// TwinCAT 3 PLC project PLC_to_Cpp
// ProgramVersion: 3.1.4023.0
// libraries:
//   Tc2_Standard, * (Beckhoff Automation GmbH)
//   Tc2_System, * (Beckhoff Automation GmbH)
//   Tc2_Utilities, * (Beckhoff Automation GmbH)
//   Tc3_IotBase, * (Beckhoff Automation GmbH)
//   Tc3_Module, * (Beckhoff Automation GmbH)
// project tree:
//   DUTs/ Cartesian.TcDUT, Joints.TcDUT, RobotState.TcDUT, RsiIncomingMsg.TcDUT, RsiOutputMsg.TcDUT
//   POUs/ FB_Rsi.TcPOU, MAIN.TcPOU, MQTTClient_Joints.TcPOU, MQTTClient_RobotState.TcPOU, MQTT_Publisher.TcPOU, MQTT_Subscriber.TcPOU, SampleUdpServer.TcPOU
//   / Task_1.TcTTO, Task_2.TcTTO

CONFIGURATION PLC_to_Cpp
    RESOURCE PLC ON TwinCAT3
        TASK Task_1(INTERVAL := T#10ms, PRIORITY := 1);
        TASK Task_2(INTERVAL := T#10ms, PRIORITY := 2);
        PROGRAM MAIN WITH Task_1 : MAIN;
        PROGRAM MQTT_Subscriber WITH Task_2 : MQTT_Subscriber;
        PROGRAM MQTT_Publisher WITH Task_2 : MQTT_Publisher;
    END_RESOURCE
END_CONFIGURATION

// ---- DUTs/Cartesian.TcDUT
TYPE Cartesian :
STRUCT
	x : LREAL :=0;
	y : LREAL :=0;
	z : LREAL :=0;
	rot1 : LREAL :=0;
	rot2 : LREAL :=0;
	rot3 : LREAL :=0;
END_STRUCT
END_TYPE

// ---- DUTs/Joints.TcDUT
TYPE Joints :
STRUCT
	joint1 : LREAL := 0;
	joint2 : LREAL := 0;
	joint3 : LREAL := 0;
	joint4 : LREAL := 0;
	joint5 : LREAL := 0;
	joint6 : LREAL := 0;
	external_axis1 : LREAL := 0;
END_STRUCT
END_TYPE

// ---- DUTs/RobotState.TcDUT
TYPE RobotState :
STRUCT
	joints_position : Joints;
	cartesian_position : Cartesian;
	joints_setpoint : Joints;
	cartesian_setpoint : Cartesian;
END_STRUCT
END_TYPE

// ---- DUTs/RsiIncomingMsg.TcDUT
TYPE RsiIncomingMsg :
STRUCT
END_STRUCT
END_TYPE

// ---- DUTs/RsiOutputMsg.TcDUT
TYPE RsiOutputMsg :
STRUCT
END_STRUCT
END_TYPE

// ---- POUs/MAIN.TcPOU
PROGRAM MAIN
VAR
	//msg : STRING(1024) := '<Rob TYPE="KUKA">\n<AIPos A1="1" A2="0.2" A3="0.3" A4="0.4" A5="0.5" A6="0.6"/>\n<ASPos A1="1.1" A2="1.2" A3="1.3" A4="1.4" A5="1.5" A6="1.6"/>\n<RIst X="100" Y="200" Z="300" A="1" B="2" C="3" />\n<RSol X="101" Y="201" Z="301" A="11" B="21" C="31" />\n<IPOC>123456789</IPOC>\n</Rob>';
					
	udp1 : SampleUdpServer;

	
END_VAR


udp1();


(*ADSLOGSTR(	msgCtrlMask:=ADSLOG_MSGTYPE_ERROR,
			msgFmtStr:='%s',
			strArg:=output_msg);
*)

END_PROGRAM

// ---- POUs/SampleUdpServer.TcPOU
{attribute 'c++_compatible'}
FUNCTION_BLOCK SampleUdpServer IMPLEMENTS ITcIoUdpProtocolRecv
VAR_INPUT
END_VAR
VAR_OUTPUT
END_VAR
VAR
    {attribute 'TcInitSymbol'}
    oid:              OTCID; 
    ipUdp:            ITcIoUdpProtocol;
    nUdpPort:         UINT := 10000;
    nReceivedPakets:  UINT;
    hrInit :          HRESULT;
    hrSend :          HRESULT;
	
	fbRsi : FB_Rsi(	sObjName:='CRsi:fbRsi',
					eObjState:=TCOM_STATE.TCOM_STATE_OP);
	output_msg : STRING(1024);
	
	robot_state AT %Q* : RobotState;
	joints_command AT %I* : Joints;
END_VAR

IF ipUdp <> 0 THEN
    ipUdp.CheckReceived();
END_IF

{attribute 'conditionalshow'}
METHOD FB_exit : BOOL
VAR_INPUT
	bInCopyCode : BOOL; // if TRUE, the exit method is called for exiting an instance that is copied afterwards (online change).
END_VAR
IF (NOT bInCopyCode AND ipUdp <> 0) THEN //Shutdown
     ipUdp.UnregisterReceiver(nUdpPort);
    FW_SafeRelease(ADR(ipUdp));
     FB_exit := TRUE;
ELSE
     FB_exit := FALSE;
END_IF
END_METHOD

{attribute 'conditionalshow'}
METHOD FB_init : BOOL
VAR_INPUT
	bInitRetains : BOOL; // if TRUE, the retain variables are initialized (warm start / cold start)
	bInCopyCode : BOOL;  // if TRUE, the instance afterwards gets moved into the copy code (online change)
END_VAR

VAR
    ipSrv: ITComObjectServer;
END_VAR
IF NOT bInCopyCode THEN
	IF ipUdp = 0 AND oid <> 0 THEN
		hrInit := FW_ObjMgr_GetObjectInstance(	oid:=oid,  
												iid:=TC_GLOBAL_IID_LIST.IID_ITcIoUdpProtocol, 
												pipUnk:=ADR(ipUdp) );
        IF SUCCEEDED(hrInit) THEN 
            IF SUCCEEDED(ipUdp.RegisterReceiver(nUdpPort, THIS^)) THEN //open port
                FB_init := TRUE;
            ELSE 
                FB_init := FALSE; 
                FW_SafeRelease(ADR(ipUdp));
            END_IF
        END_IF
    ELSIF oid = 0 THEN 
        FB_init := FALSE; 
        hrInit := ERR_INVALID_PARAM;                 
    END_IF
END_IF
END_METHOD

{attribute 'conditionalshow'}
METHOD FB_reinit : BOOL
VAR_INPUT
END_VAR
IF (ipUdp <> 0) THEN 
 ipUdp.RegisterReceiver(nUdpPort, THIS^);
END_IF
END_METHOD

{attribute 'object_name' := 'ReceiveData'}
{attribute 'c++_compatible'}
{attribute 'signature_flag' := '33554688'}
{attribute 'pack_mode' := '4'}
{attribute 'show'}
{attribute 'minimal_input_size' := '4'}
METHOD ReceiveData : HRESULT
VAR_INPUT
	ipAddr	: UDINT;
	udpDestPort	: UINT;
	udpSrcPort	: UINT;
	nData	: UDINT;
	pData	: PVOID;
	pVlan	: POINTER TO ETYPE_VLAN_HEADER := 0;
END_VAR

VAR
	msg_length : UINT;
END_VAR
nReceivedPakets := nReceivedPakets+1;
IF ipUdp <> 0 THEN
	
	IF fbRsi.ip <> 0 THEN
	
	
	//	fbRsi.ip.read_incoming_msg(msg);
	//	fbRsi.set_string(msg);
		fbRsi.ip.read_incoming_msg(nData, pData);
		robot_state.joints_position.joint1 := fbRsi.ip.get_axis_1();
		robot_state.joints_position.joint2 := fbRsi.ip.get_axis_2();
		robot_state.joints_position.joint3 := fbRsi.ip.get_axis_3();
		robot_state.joints_position.joint4 := fbRsi.ip.get_axis_4();
		robot_state.joints_position.joint5 := fbRsi.ip.get_axis_5();
		robot_state.joints_position.joint6 := fbRsi.ip.get_axis_6();
		robot_state.joints_position.external_axis1 := fbRsi.ip.get_external_axis_1();
	
		robot_state.joints_setpoint.joint1 := fbRsi.ip.get_axis_1_setpoint();
		robot_state.joints_setpoint.joint2 := fbRsi.ip.get_axis_2_setpoint();
		robot_state.joints_setpoint.joint3 := fbRsi.ip.get_axis_3_setpoint();
		robot_state.joints_setpoint.joint4 := fbRsi.ip.get_axis_4_setpoint();
		robot_state.joints_setpoint.joint5 := fbRsi.ip.get_axis_5_setpoint();
		robot_state.joints_setpoint.joint6 := fbRsi.ip.get_axis_6_setpoint();
		robot_state.joints_setpoint.external_axis1 := fbRsi.ip.get_external_axis_1_setpoint();
		
		robot_state.cartesian_position.x := fbRsi.ip.get_cartesian_x();
		robot_state.cartesian_position.y := fbRsi.ip.get_cartesian_y();
		robot_state.cartesian_position.z := fbRsi.ip.get_cartesian_z();
		robot_state.cartesian_position.rot1 := fbRsi.ip.get_cartesian_rot1();
		robot_state.cartesian_position.rot2 := fbRsi.ip.get_cartesian_rot2();
		robot_state.cartesian_position.rot3 := fbRsi.ip.get_cartesian_rot3();
		
		robot_state.cartesian_setpoint.x := fbRsi.ip.get_cartesian_x_setpoint();
		robot_state.cartesian_setpoint.y := fbRsi.ip.get_cartesian_y_setpoint();
		robot_state.cartesian_setpoint.z := fbRsi.ip.get_cartesian_z_setpoint();
		robot_state.cartesian_setpoint.rot1 := fbRsi.ip.get_cartesian_rot1_setpoint();
		robot_state.cartesian_setpoint.rot2 := fbRsi.ip.get_cartesian_rot2_setpoint();
		robot_state.cartesian_setpoint.rot3 := fbRsi.ip.get_cartesian_rot3_setpoint();
		
		msg_length:= fbRsi.ip.write_msg(SIZEOF(output_msg),
										ADR(output_msg), 
										joints_command.joint1, 
										joints_command.joint2, 
										joints_command.joint3, 
										joints_command.joint4, 
										joints_command.joint5, 
										joints_command.joint6,
										joints_command.external_axis1);
	
	
		hrSend := ipUdp.SendData(	ipAddr, 
									udpSrcPort, 
									udpDestPort, 
									msg_length, 
									ADR(output_msg), 
									TRUE, 
									0); // send data back

	END_IF
END_IF
END_METHOD

{attribute 'object_name' := 'TcAddRef'}
{attribute 'c++_compatible'}
{attribute 'signature_flag' := '33554688'}
{attribute 'pack_mode' := '4'}
{attribute 'show'}
{attribute 'minimal_input_size' := '4'}
METHOD TcAddRef : UDINT
END_METHOD

{attribute 'object_name' := 'TcQueryInterface'}
{attribute 'c++_compatible'}
{attribute 'signature_flag' := '33554688'}
{attribute 'pack_mode' := '4'}
{attribute 'show'}
{attribute 'minimal_input_size' := '4'}
METHOD TcQueryInterface : HRESULT
VAR_INPUT
	iid	: REFERENCE TO IID;
	pipItf	: POINTER TO PVOID;
END_VAR

VAR
    ipUdpRecv : ITcIoUdpProtocolRecv;
    ipUnknown : ITcUnknown;    
END_VAR
IF GuidsEqual(ADR(iid), ADR(TC_GLOBAL_IID_LIST.IID_ITcIoUdpProtocolRecv)) THEN
    ipUdpRecv := THIS^; // cast to interface pointer
    pipItf^ := ITCUNKNOWN_TO_PVOID(ipUdpRecv);
    TcAddRef();
    TcQueryInterface := S_OK;
ELSIF GuidsEqual(ADR(iid), ADR(TC_GLOBAL_IID_LIST.IID_ITcUnknown)) THEN
    ipUnknown := THIS^; // cast to interface pointer
    pipItf^ := ITCUNKNOWN_TO_PVOID(ipUnknown);
    TcAddRef();
    TcQueryInterface := S_OK;
ELSE
    TcQueryInterface := E_HRESULTAdsErr.NOINTERFACE ; //Call super if this fb extends some other
END_IF
END_METHOD

{attribute 'object_name' := 'TcRelease'}
{attribute 'c++_compatible'}
{attribute 'signature_flag' := '33554688'}
{attribute 'pack_mode' := '4'}
{attribute 'show'}
{attribute 'minimal_input_size' := '4'}
METHOD TcRelease : UDINT
END_METHOD

END_FUNCTION_BLOCK

// ---- POUs/FB_Rsi.TcPOU
FUNCTION_BLOCK FB_Rsi

VAR_OUTPUT
	 ip : IRsi;
END_VAR

VAR;
	objName : STRING;
	classid : CLSID := STRING_TO_GUID('eb745b26-c68e-4ee7-9e8f-1d06260b78a8');
	iid : IID := TC_GLOBAL_IID_LIST.IID_IRsi;
	hrInit : HRESULT;
END_VAR

METHOD FB_exit : BOOL
VAR_INPUT
	bInCopyCode : BOOL; // if TRUE, the exit method is called for exiting an instance that is copied afterwards (online change).
END_VAR
IF	NOT bInCopyCode THEN
	FW_ObjMgr_DeleteInstance(ADR(ip));
END_IF
END_METHOD

METHOD FB_init : BOOL
VAR_INPUT
	bInitRetains : BOOL; // if TRUE, the retain variables are initialized (warm start / cold start)
	bInCopyCode : BOOL;  // if TRUE, the instance afterwards gets moved into the copy code (online change)

	sObjName: STRING;
	eObjState: TCOM_STATE;
END_VAR
objName:=sObjName;
hrInit:= FW_ObjMgr_CreateAndInitInstance(	clsId:=classId,
											iid:=iid,
											pipUnk:=ADR(ip),
											objId:=OTCID_CreateNewId,
											parentId:=TwinCAT_SystemInfoVarList._AppInfo.ObjId,
											name:=sObjName,
											state:=eObjState,
											pInitData:=0);
END_METHOD

END_FUNCTION_BLOCK

// ---- POUs/MQTT_Subscriber.TcPOU
PROGRAM MQTT_Subscriber
VAR
	
	received_msg_size : UDINT;
	sTopicSub : STRING;
	eQoSSub : TcIotMqttQos;
	bConnectSub : BOOL;
	MQTT_client : MQTTClient_Joints;	
	isConnected : BOOL;
	isSub : BOOL;
	
	joints_command AT %Q* : Joints;
	incoming_msg AT %I* : Joints;
END_VAR

sTopicSub := 'robot1/command'; 
eQoSSub := 1;
bConnectSub := TRUE;
isConnected := MQTT_client.bConnected;
MQTT_client.sHostName := '169.254.252.101';

//SUBSCRIBE
MQTT_client.Execute(bConnectSub);
isSub := MQTT_client.Subscribe(	sTopic := sTopicSub, 
								eQoS := eQoSSub);
incoming_msg := MQTT_client.sPayloadRcv;

joints_command := incoming_msg;

END_PROGRAM

// ---- POUs/MQTTClient_Joints.TcPOU
{attribute 'c++_compatible'}
FUNCTION_BLOCK MQTTClient_Joints EXTENDS FB_IotMqttClient
VAR_INPUT
	{attribute 'TcEncoding':='UTF-8'}
	 sTopicRcv   : STRING(255);
	 {attribute 'TcEncoding':='UTF-8'}
	 sPayloadRcv : Joints;
END_VAR
VAR_OUTPUT
END_VAR
VAR
END_VAR

{attribute 'c++_compatible'}
{attribute 'pack_mode' := '4'}
{attribute 'show'}
{attribute 'minimal_input_size' := '4'}
METHOD OnMqttMessage : HRESULT
VAR_IN_OUT CONSTANT
    topic    : STRING;
END_VAR
VAR_INPUT
    payload  : PVOID;
    length   : UDINT;
    qos      : TcIotMqttQos;
    repeated : BOOL;
END_VAR
VAR
    nPayloadRcvLen : UDINT;
END_VAR
STRNCPY( ADR(sTopicRcv), ADR(topic), SIZEOF(sTopicRcv) );
nPayloadRcvLen := MIN(length, DINT_TO_UDINT(SIZEOF(sPayloadRcv)));
MEMCPY( ADR(sPayloadRcv), payload, nPayloadRcvLen );

OnMqttMessage := S_OK;
END_METHOD

END_FUNCTION_BLOCK

// ---- POUs/MQTT_Publisher.TcPOU
PROGRAM MQTT_Publisher
VAR
	robot_state AT %I* : RobotState;
	robot_state_msg AT %Q* : RobotState;
	
	received_msg_size : UDINT;
	PayloadPub : PVOID;
	PayloadSizePub : UDINT;
	sTopicPub : STRING := 'robot1/state';
	eQoSPub : TcIotMqttQos;
	bConnectPub : BOOL;
	MQTT_client : MQTTClient_RobotState;	
	bRetainPub : BOOL;
	bQueuePub : BOOL;
	isConnected : BOOL;
	isPub : BOOL;
	
	
	// Only for test putpose
	joints_command_fake AT %Q* : Joints;
	MQTT_client_fake : MQTTClient_Joints;
	
END_VAR

bRetainPub := FALSE; 
bQueuePub := FALSE;
bConnectPub := TRUE;
isConnected := MQTT_client.bConnected;
MQTT_client.sHostName := '169.254.252.101';

robot_state_msg := robot_state;

PayloadPub := ADR(robot_state_msg);
PayloadSizePub := SIZEOF(robot_state_msg);
MQTT_client.Execute(bConnect := bConnectPub);
isPub := MQTT_client.Publish(	sTopic := sTopicPub, 
								pPayload := PayloadPub, 
								nPayloadSize := PayloadSizePub, 
								eQos := eQoSPub, 
								bRetain := bRetainPub, 
								bQueue := bQueuePub);
isConnected := MQTT_client.bConnected;

// Only for test purpose
(*
joints_command_fake.joint1 := -0.01;
joints_command_fake.joint2 := -0.02;
joints_command_fake.joint3 := -0.03;
joints_command_fake.joint4 := -0.04;
joints_command_fake.joint5 := -0.05;
joints_command_fake.joint6 := -0.010;
joints_command_fake.external_axis1 := -0.001;

PayloadPub := ADR(joints_command_fake);
PayloadSizePub := SIZEOF(joints_command_fake);
MQTT_client_fake.sHostName := MQTT_client.sHostName;
MQTT_client_fake.Execute(bConnect := bConnectPub);
MQTT_client_fake.Publish(	sTopic := 'robot1/command', 
												pPayload := PayloadPub, 
												nPayloadSize := PayloadSizePub, 
												eQos := eQoSPub, 
												bRetain := bRetainPub, 
												bQueue := bQueuePub);
*)

END_PROGRAM

// ---- POUs/MQTTClient_RobotState.TcPOU
{attribute 'c++_compatible'}
FUNCTION_BLOCK MQTTClient_RobotState EXTENDS FB_IotMqttClient
VAR_INPUT
	{attribute 'TcEncoding':='UTF-8'}
	 sTopicRcv   : STRING(255);
	 {attribute 'TcEncoding':='UTF-8'}
	 sPayloadRcv : RobotState;
END_VAR
VAR_OUTPUT
END_VAR
VAR
END_VAR

{attribute 'c++_compatible'}
{attribute 'pack_mode' := '4'}
{attribute 'show'}
{attribute 'minimal_input_size' := '4'}
METHOD OnMqttMessage : HRESULT
VAR_IN_OUT CONSTANT
    topic    : STRING;
END_VAR
VAR_INPUT
    payload  : PVOID;
    length   : UDINT;
    qos      : TcIotMqttQos;
    repeated : BOOL;
END_VAR
VAR
    nPayloadRcvLen : UDINT;
END_VAR
STRNCPY( ADR(sTopicRcv), ADR(topic), SIZEOF(sTopicRcv) );
nPayloadRcvLen := MIN(length, DINT_TO_UDINT(SIZEOF(sPayloadRcv)));
MEMCPY( ADR(sPayloadRcv), payload, nPayloadRcvLen );

OnMqttMessage := S_OK;
END_METHOD

END_FUNCTION_BLOCK
